// TIA Portal V18 export
// export: Created 2025-12-01T17:50:32.4744177Z, ExportSetting None, DisplayName Totally Integrated Automation Portal, DisplayVersion V18 Update 5, DisplayName TIA Portal Openness, DisplayVersion V18 Update 5, DisplayName TIA Portal Teamcenter Gateway, DisplayVersion V18, DisplayName TIA Portal Version Control Interface, DisplayVersion V18, DisplayName STEP 7 Professional, DisplayVersion V18 Update 5, DisplayName STEP 7 Safety, DisplayVersion V18, DisplayName WinCC Professional, DisplayVersion V18 Update 5
FUNCTION_BLOCK "FB_Keyence_SR1000"   // FB1230, SCL
{ S7_Optimized_Access := 'TRUE' }
// stored: AutoNumber false, MemoryReserve 100, SetENOAutomatically false
   VAR_INPUT
      "I_Handshake and Genera_InAdr" : HW_IO;
      I_BUSYStatusBits_InAdr : HW_IO;
      I_CompletionStatus_InAdr : HW_IO;
      I_ErrorStatusBits_InAdr : HW_IO;
      "I_Terminal Status InAdr" : HW_IO;
      "I_Unstable Read Status Bits_InAdr" : HW_IO;
      "I_Matching Level and Total_InAdr" : HW_IO;
      "I_Operation Result Status InAdr" : HW_IO;
      "I_Read Data 128Byte InAdr" : HW_IO;
      "I_Latch and Error OutAdr" : HW_IO;
      "I_Operation instruction_OutAdr" : HW_IO;
      "I_Completion OutAdr" : HW_IO;
      "I_Parameter Bank Number_OutAdr" : HW_IO;
      "I_User Data 128Byte_OutAdr" : HW_IO;
   END_VAR
   VAR_OUTPUT
      io_nError : Int;
      io_nWarning : Int;
   END_VAR
   VAR_IN_OUT
      IO_udtData : "ST_KeyenceSR1000";
   END_VAR
   VAR
      s_nValue : Array[0..20] of Int;
      sUP : Array[0..10] of R_TRIG;
      TON { S7_SetPoint := 'True'} : Array[0..10] of TON_TIME;
      FB_Step { S7_SetPoint := 'True'} : "FB_Step";
      sPN_IN : Struct
         Handshake : Byte;
         BUSYStatusBits : Byte;
         CompletionStatus : Byte;
         ErrorStatusBits : Byte;
         TerminalStatus : Byte;
         UnstableReadStatusBits : Byte;
         MatchingLevelandTotal : Array[1..8] of Byte;
         OperationResultStatus : Array[1..20] of Byte;
         ReadData128Byte : Array[1..136] of Byte;
      END_STRUCT;
      sPN_Out : Struct
         LatchErrorClear : Byte;   // Latch and Error Clear Control Bits
         OperationInstruction : Byte;   // Operation instruction Control Bits
         Completion : Byte;   // Completion Clear Control Bits
         ParBankNo : Array[1..2] of Byte;   // Parameter Bank Number
         UserData128byte : Array[1..136] of Byte;   // UserData128byte
      END_STRUCT;
      Flag : Array[0..10] of Bool;
   END_VAR
   VAR_TEMP
      tInt : Array[1..8] of Int;
      i : Int;
      TempBytes : Array[1..128] of Char;
   END_VAR
BEGIN
   REGION Read PN Data 读取PN数据
       // 插槽1
       #s_nValue[1] := DPRD_DAT(LADDR := #"I_Handshake and Genera_InAdr",
                                RECORD => #sPN_IN.Handshake);
       //插槽2
       #s_nValue[2] := DPRD_DAT(LADDR := #I_BUSYStatusBits_InAdr,
                                RECORD => #sPN_IN.BUSYStatusBits);
       //插槽3
       #s_nValue[3] := DPRD_DAT(LADDR := #I_CompletionStatus_InAdr,
                                RECORD => #sPN_IN.CompletionStatus);
       //插槽4
       #s_nValue[4] := DPRD_DAT(LADDR := #I_ErrorStatusBits_InAdr,
                                RECORD => #sPN_IN.ErrorStatusBits);
       //插槽5
       #s_nValue[5] := DPRD_DAT(LADDR := #"I_Terminal Status InAdr",
                                RECORD => #sPN_IN.TerminalStatus);
       //插槽6
       #s_nValue[6] := DPRD_DAT(LADDR := #"I_Unstable Read Status Bits_InAdr",
                                RECORD => #sPN_IN.UnstableReadStatusBits);
       //插槽7
       #s_nValue[7] := DPRD_DAT(LADDR := #"I_Matching Level and Total_InAdr",
                                RECORD => #sPN_IN.MatchingLevelandTotal);
       //插槽8
       #s_nValue[8] := DPRD_DAT(LADDR := #"I_Operation Result Status InAdr",
                                RECORD => #sPN_IN.OperationResultStatus);
       //插槽9
       #s_nValue[9] := DPRD_DAT(LADDR := #"I_Read Data 128Byte InAdr",
                                RECORD => #sPN_IN.ReadData128Byte);

   END_REGION

   REGION CopyReadData()
       //************************************************************************************************
       //分配输入数据(控制数据解析)/Asignment of the input data (control word)
       //************************************************************************************************
       #IO_udtData.In.bBusy := #sPN_IN.BUSYStatusBits.%X1;
       #IO_udtData.In.bError := #sPN_IN.Handshake.%X0;
       #IO_udtData.In.bReadComplete := #sPN_IN.CompletionStatus.%X0;
       #IO_udtData.In.bReadFailure := #sPN_IN.ErrorStatusBits.%X0;
       #IO_udtData.In.nReadResultCode := #sPN_IN.OperationResultStatus[4];

   END_REGION

   REGION Error Code 报错信息
       //流程超时/Process overtime alarm   X0
       #TON[1](IN := #IO_udtData.Common.nMode <> 0,
               PT := T#12S);
       IF #TON[1].Q THEN
           #IO_udtData.Common.nErrorNo := 1;
           #io_nError.%X0 := 1;
       END_IF;

       //读码超时

       #TON[2](IN := NOT #FB_Step.sCondition AND #FB_Step.sNextNo = 1100,
               PT := T#8S);

       //错误标志/Error flag
       //
       IF #IO_udtData.Common.nErrorNo <> 0 THEN
           #IO_udtData.Common.bError := TRUE;
           #IO_udtData.Common.nMode := 0;
       END_IF;

       //复位报警信息/Reset alarm messages
       IF #IO_udtData.Common.bReset AND #IO_udtData.Common.bError THEN
           #IO_udtData.Common.nErrorNo := 0;
           #io_nError := 0;
           #IO_udtData.Common.bError := FALSE;
       END_IF;
       //报警复位
       #IO_udtData.Out.bErrorClear := #IO_udtData.Common.bReset;

   END_REGION

   REGION 提示信息
       // Statement section REGION
       #IO_udtData.Common.nWarningNo := #IO_udtData.In.nReadResultCode;
   END_REGION


   REGION Data 读码数据解析
       IF #IO_udtData.In.bReadComplete THEN
           #IO_udtData.In.nDataSize := #sPN_IN.ReadData128Byte[8] - 1;
           FOR #i := 1 TO 128 DO
               #IO_udtData.In.aData[#i] := #sPN_IN.ReadData128Byte[#i + 8];
           END_FOR;
           Chars_TO_Strg(Chars := #IO_udtData.In.aData,
                         pChars := 0,
                         Cnt := #IO_udtData.In.nDataSize,
                         Strg => #IO_udtData.RecordCode);
       END_IF;
   END_REGION

   REGION AutoStep
       #FB_Step(1);
       IF #IO_udtData.Common.nMode <> 0 THEN
           CASE #FB_Step.sCurrNo OF
               0:
                   #FB_Step.sCondition := #IO_udtData.Common.nMode = 1;
                   #FB_Step.sNextNo := 1000;
               1000://开始读取
                   IF #FB_Step.sPls THEN
                       #IO_udtData.Out.bReadRequest := 1;
                       #IO_udtData.RecordCode := '';
                       #IO_udtData.In.aData := #TempBytes;
                       #IO_udtData.In.nDataSize := 0;
                       #IO_udtData.Common.bDone := 0;
                       #IO_udtData.Common.bNG := 0;
                       #IO_udtData.Common.bOK := 0;
                   END_IF;
                   #FB_Step.sCondition := #IO_udtData.In.bBusy;
                   #FB_Step.sNextNo := 1100;
               1100://等待读取完成

                   #FB_Step.sDealyTime := T#10MS;

                   #FB_Step.sCondition :=( #IO_udtData.In.bReadComplete AND NOT #IO_udtData.In.bBusy ) OR #TON[2].Q;
                   IF #FB_Step.sCondition THEN
                       #IO_udtData.Out.bReadRequest := 0;
                   END_IF;
                   #FB_Step.sNextNo := 1200;
               1200://判断读取结果
                   IF #IO_udtData.RecordCode = 'ERROR' THEN
                       #IO_udtData.Common.bNG := 1;//读取NG
                       #IO_udtData.Common.bOK := 0;
                   ELSE
                       #IO_udtData.Common.bNG := 0;
                       #IO_udtData.Common.bOK := 1;//读取OK
                   END_IF;
                   #FB_Step.sCondition := 1;
                   #FB_Step.sNextNo := 1300;
               1300://读取完成
                   IF #FB_Step.sPls THEN
                       #IO_udtData.Out.bReadComlpleteClear := 1;
                   END_IF;
                   #FB_Step.sCondition := NOT #IO_udtData.In.bReadComplete AND NOT #IO_udtData.In.bReadFailure;
                   #FB_Step.sNextNo := 1400;
               1400://
                   IF #FB_Step.sPls THEN
                       #IO_udtData.Out.bReadComlpleteClear := 0;
                       #IO_udtData.Common.bDone := 1;
                       #IO_udtData.Common.nMode := 0;
                   END_IF;
                   #FB_Step.sCondition := 1;
                   #FB_Step.sNextNo := 0;
           END_CASE;
       ELSE
           #FB_Step.sCurrNo := 0;
           #IO_udtData.Out.bReadComlpleteClear := 0;
           #IO_udtData.Out.bReadRequest := 0;
       END_IF;
   END_REGION

   REGION CopyWriteData()   
       //************************************************************************************************
       //分配输出数据(控制数据解析)/Asignment of the output data (control word)
       //************************************************************************************************
       #sPN_Out.OperationInstruction.%X0 := #IO_udtData.Out.bReadRequest;
       #sPN_Out.LatchErrorClear.%X7:= #IO_udtData.Out.bErrorClear;
       #sPN_Out.Completion.%X0 := #IO_udtData.Out.bReadComlpleteClear;



   END_REGION

   REGION Write Data 写入PN数据
       // 插槽10
       #s_nValue[10] := DPWR_DAT(LADDR := #"I_Latch and Error OutAdr",
                                RECORD := #sPN_Out.LatchErrorClear);
       // 插槽11
       #s_nValue[11] := DPWR_DAT(LADDR := #"I_Operation instruction_OutAdr",
                                RECORD := #sPN_Out.OperationInstruction);
       //插槽12
      #s_nValue[12] := DPWR_DAT(LADDR := #"I_Completion OutAdr",
                                RECORD := #sPN_Out.Completion);
       // 插槽13
      #s_nValue[13] := DPWR_DAT(LADDR := #"I_Parameter Bank Number_OutAdr",
                                RECORD := #sPN_Out.ParBankNo);
       // 插槽14
       #s_nValue[14] := DPWR_DAT(LADDR := #"I_User Data 128Byte_OutAdr",
                                RECORD := #sPN_Out.UserData128byte);
   END_REGION
END_FUNCTION_BLOCK
